//==============================================================
// 五盘阻尼器上下料主流程
//
// 一个bStart上升沿按Tray启动时冻结的物理层计划处理料盘，每盘4行×6列。
//
// 当前测试版本：
// 1. DamperX、DamperY在同一扫描周期启动；
// 2. 分别锁存X、Y完成信号，全部到位后继续；
// 3. 夹爪步骤直接通过；
// 4. 转台使用轴8在0°/180°之间绝对位置交替运动；
// 5. 夹紧轴使用位置模式模拟夹紧；
// 6. 调整过程由FB_TurntableProcess使用3秒TON模拟；
// 7. 换盘过程使用3秒TON模拟；
// 8. XY/Z/Rotation独立监督；统一Process Fault接入整机Stop链。
//==============================================================

FUNCTION_BLOCK FB_DamperProcess

VAR_INPUT
	
	bGripperActionDone  : BOOL; // 上一扫描至本扫描的动作FB结果
	bGripperActionError : BOOL;
    bGripperCloseTargetReachedWithoutGrip : BOOL;
    bGripperActionReady : BOOL; // Action Idle且Manager/Control均已释放
    // FALSE变为TRUE时启动完整五盘循环。
    bStart : BOOL;

    // 调试时产生上升沿，重新计算料位、备料位和缓冲位坐标。
    // 正常自动运行期间不要触发。
    bReinitializeCoordinates : BOOL;
	
	// 来自转台协调FB；由于MAIN先调用本FB，这里读取上一扫描周期状态。
    stTurntableStatus : ST_DamperTurntableStatus;
	// 当前料盘已经到达阻尼器取料位置。
	bTrayAtDamperPosition : BOOL;
	
	// 一次换盘已经完成，新料盘到达工作位置。
	// 保持到本FB撤销bTrayChangeRequest。
	bTrayChangeDone : BOOL;
	
	// 当前位于阻尼器工作位置的实际料盘层号。
	nTrayAtDamperLayer : INT;
    bCurrentTrayIsLastPlanned : BOOL; // Tray转接：当前工作位置料盘是固定计划最终盘
	// TRUE：立即中止本轮阻尼器自动流程。
	// 不清空料位、备料位、调整位和缓冲位物料状态。
	bAbort : BOOL;
    bReset : BOOL; // 复用整机故障复位
	// TRUE表示整机准备FB已经完成Z=110、XY=(1,1)、Rotation=0。
	bMachinePrepared : BOOL;
END_VAR

VAR_IN_OUT
    stAxisX : ST_AxisInterface; // DamperX：行方向
    stAxisY : ST_AxisInterface; // DamperY：列方向
    stAxisZ : ST_AxisInterface; // DamperZ：升降方向
	
	// 阻尼器夹爪旋转轴，对应统一轴数组第6轴。
    stAxisRotation : ST_AxisInterface;
END_VAR

VAR_OUTPUT
    bError : BOOL;
    uiErrorAxis : UINT;
    udiErrorCode : UDINT;
    bBusy : BOOL;
    bDone : BOOL;
    bCurrentTrayDone : BOOL;
    bTrayChangeRequest : BOOL;
    bInitialized : BOOL;
	
    //==========================================================
    // Damper三轴自动流程启动预定位完成
    //
    // TRUE表示：
    // 1. DamperZ已经位于110mm安全高度；
    // 2. DamperX/Y已经位于(1,1)料位上方；
    // 3. Tray机构可以开始取第一盘。
    //==========================================================
    bPrePositionDone : BOOL;

    // 最近一次螺钉角度视觉事务诊断。
    bVisionFault : BOOL;
    // 为兼容现有监控符号保留；本版本不再生成或使用Fallback结果。
    bVisionFallbackUsed : BOOL;
    eVisionError : E_VisionError := E_VisionError.None;

    // 发送给FB_TurntableProcess的保持型请求。
    stTurntableInput : ST_DamperTurntableInput;
    // 最近一次完成调整的料盘编号。
    nLastCompletedTray : INT;

    nCurrentTray   : INT;
    nCurrentRow    : INT;
    nCurrentColumn : DINT;

//==============================================================
// 上一件阻尼器的原始取料位置
//
// 用途：
// 1. 阻尼器取走后，原料位临时显示Adjusting；
// 2. 阻尼器放到其他实际位置后，将仍为Adjusting的原料位清空；
// 3. 如果原料位已经被其他合格品占用，则不能错误清空。
//==============================================================
	nPreviousSourceTray   : INT;
	nPreviousSourceRow    : INT;
	nPreviousSourceColumn : DINT;

    eCurrentStep : E_DamperProcessStep;
    eTakeStep    : E_DamperTakeStep;
    ePlaceStep   : E_DamperPlaceStep;

    // 当前工作位置料盘的数据。
    aSlots : A_DamperSlotGrid;

    // 转台两个位置及最终缓冲位的内容状态。
    eTransferPositionState   : E_DamperSlotState;
    eAdjustmentPositionState : E_DamperSlotState;
    eBufferPositionState     : E_DamperSlotState;

    // 公共工作位置，单位mm。
    fTrayPickZ     : LREAL;
    fTraySafeZ     : LREAL;
    fTransferX     : LREAL;
    fTransferY     : LREAL;
    fTransferPickZ : LREAL;
    fTransferSafeZ : LREAL;
    fBufferX       : LREAL;
    fBufferY       : LREAL;
    fBufferPickZ   : LREAL;
    fBufferSafeZ   : LREAL;
	
	bGripperActionExecute : BOOL; // 给COM3动作FB的保持型请求
	eGripperActionCommand : E_GripperCommand;
    bGripperAllowCloseTargetWithoutGrip : BOOL;
END_VAR

VAR
    trigStart : R_TRIG;
    fbXYMotionTimeout : TON;
    fbZMotionTimeout : TON;
    fbRotationMotionTimeout : TON;
    trigReinitializeCoordinates : R_TRIG;
	
    //==========================================================
    // 料盘坐标参数
    //==========================================================





    //==========================================================
    // Z轴参数
    //==========================================================

	//==========================================================
	// Z轴统一抬升绝对位置
	//
	// 所有XY运动前，以及取放料完成后，Z轴均抬升到110mm。
	// 该位置是实际测量确认的安全位置，不再进行高度计算。
	//==========================================================

	
	//==========================================================
	// 转台备料位实测绝对坐标，单位mm
	//==========================================================


	
	
	//==========================================================
	// 最终缓冲位1绝对坐标
	//
	// 当前为临时模拟值。
	// 实测完成后只修改以下三个参数。
	//==========================================================



	
    //==========================================================
    // 测试运动参数
    //==========================================================




    // 判断某根XY轴是否已经在目标位置。


		
    //==========================================================
    // 主流程内部变量
    //==========================================================
    bCoordinatesInitialized : BOOL;
    bPreviousPartAvailable  : BOOL;
    // 单槽位内部结果：只推进搜索，不代表实际取料成功。
    bTakeSkippedNoScrew : BOOL;
    bTakeSkippedEmptySlot : BOOL; // 物理空位已Open并回安全Z，独立于视觉Skip

    fCurrentSlotX : LREAL;
    fCurrentSlotY : LREAL;

    //==========================================================
    // XY并行运动内部状态
    //==========================================================
    bXYCommandIssued : BOOL;
    bXDoneLatched    : BOOL;
    bYDoneLatched    : BOOL;

    //==========================================================
    // Z轴运动内部状态
    //==========================================================
    bZCommandIssued : BOOL;
    bZDoneLatched   : BOOL;
	
	bWaitingTrayResult : BOOL;//等待料盘更换完成
    nTrayAwaitingResult : INT;//
    bStartPending : BOOL;//开始信号
	
	// 转台后的并行流程锁存。
	bPreviousPlaceDone       : BOOL;
	bExchangeCompleteLatched : BOOL;
	
	
	//==============================================================
	// 取料前相机检测位置参数
	//
	// 相机位于夹爪Y正方向90mm，因此相机对准阻尼器时：
	// 轴Y目标位置 = 阻尼器Y位置 - 90mm。
	//==============================================================


	
	// 当前检测高度与统一安全高度相同。

	
	
	//==============================================================
	// PLC相机检测模拟参数
	//==============================================================
	
	// 每个阻尼器到达相机位置后等待2秒。

	
	// 模拟相机返回机械零点坐标系下的绝对角度。

	
	
	//==============================================================
	// DamperRotation临时运动参数
	//
	// 单位应与DamperRotation NC轴缩放一致，当前按照“度”使用。
	//==============================================================



	
	// 修正角绝对值小于该值时，不发送旋转命令。

	
	//==============================================================
	// 二维码扫描绝对角度参数
	//
	// XY到达转台备料位后，DamperZ保持在110mm，
	// DamperRotation绝对运动到“相机角度+扫码偏移角”。
	// 当前使用旋转完成作为二维码扫描成功条件。
	//==============================================================
	//==============================================================
	// 相机检测与旋转运行变量
	//==============================================================
	
	// 螺钉角度业务视觉封装；内部拥有独立FB_VisionRequest实例。
	fbScrewAngleVision : FB_ScrewAngleVision;
	
	// 相机对准当前阻尼器时，DamperXY的目标位置。
	fCurrentVisionX : LREAL;
	fCurrentVisionY : LREAL;
	
	// 锁存原始检测角度、Python给出的机械修正量和本件实际机械基准角度。
	fDetectedAngleLatched   : LREAL;
	fCorrectionAngleLatched : LREAL;
	fRotationBaseAngle      : LREAL;
	fScanTargetAngle        : LREAL;
	bRotationCorrectionRequired : BOOL;
	
	// 防止每扫描周期重复发送DamperRotation绝对运动命令。
	bRotationCommandIssued : BOOL;
	
	//==============================================================
	// 取料后Z轴抬升与DamperRotation并行运动完成锁存
	//
	// 两根轴的完成信号可能出现在不同PLC扫描周期，
	// 因此必须分别锁存，不能直接将两个bDone进行AND判断。
	//==============================================================
	
	// 夹紧后：Z轴抬升与Rotation到相机角度的完成锁存。
	bCameraLiftZDoneLatched    : BOOL;
	bCameraRotationDoneLatched : BOOL;
	
	// 放料后：Z轴抬升、转台换位与Rotation回零的完成锁存。
	bResetLiftZDoneLatched     : BOOL;
	bResetTurntableDoneLatched : BOOL;
	bResetRotationDoneLatched  : BOOL;
END_VAR

//==============================================================
// 1. 更新输入上升沿
//==============================================================
trigStart(CLK := bStart);

trigReinitializeCoordinates(
    CLK := bReinitializeCoordinates
);

bGripperActionExecute := FALSE;
eGripperActionCommand := E_GripperCommand.None;
bGripperAllowCloseTargetWithoutGrip := FALSE;

// 机械流程只保持请求并消费统一结果；Simulation延时和ADS握手
// 均封装在FB_ScrewAngleVision中。
fbScrewAngleVision(
    bExecute := bBusy
                AND (eCurrentStep = E_DamperProcessStep.TakeCurrentDamper)
                AND (eTakeStep = E_DamperTakeStep.AcquireVisionResult),
    bCancel := bAbort OR bReset
);

//==============================================================
// 外部中止优先级最高
//==============================================================
IF bReset THEN
    bError := FALSE;
    uiErrorAxis := 0;
    udiErrorCode := TO_UDINT(E_DamperErrorCode.None);
    bVisionFault := FALSE;
    eVisionError := E_VisionError.None;
END_IF;

IF bAbort OR bReset THEN
    M_AbortProcess(
        ioAxisX := stAxisX,
        ioAxisY := stAxisY,
        ioAxisZ := stAxisZ,
        ioAxisRotation := stAxisRotation
    );

    RETURN;
END_IF;


IF trigStart.Q AND NOT bError THEN
    // 锁存一次完整五盘流程启动请求。
    bStartPending := TRUE;

    // 新一轮流程必须重新执行Damper三轴预定位。
    // 防止上一轮残留的TRUE让Tray机构提前启动。
    bPrePositionDone := FALSE;
END_IF;


	// 当前测试阶段让转台协调FB一直保持使能，先完成0°和松开位置初始化。
	// 实机后可改为系统自动模式许可。
	stTurntableInput.bEnable := bStart
								OR bStartPending
								OR bBusy;
	stTurntableInput.bAdjustmentAccepted := FALSE;
	stTurntableInput.bAdjustmentDone := FALSE;
	// 最终质量只由FB_AdjustmentProcess经协调器写入，Damper不再提供固定合格值。
	stTurntableInput.bAdjustmentQualified := FALSE;
	stTurntableInput.bTransferCaptureOK := TRUE;
	stTurntableInput.bAdjustmentCaptureOK := TRUE;
	stTurntableInput.bReset := FALSE;
//==============================================================
// 2. 首次调用或调试命令触发时初始化坐标
//
// 重新初始化坐标不会修改生产状态。
//==============================================================
IF
    (NOT bCoordinatesInitialized)
    OR
    (
        trigReinitializeCoordinates.Q
        AND NOT bBusy
    )
THEN
    M_InitializeDamperCoordinates();
    bCoordinatesInitialized := TRUE;
END_IF;


//==============================================================
// 3. 模拟换盘定时器
//
// 只有进入WaitTrayChange时定时器才开始计时。
// 离开该步骤后自动复位。
//==============================================================

//==============================================================
// 4. 清除单周期输出
//==============================================================
bCurrentTrayDone := FALSE;

// 第24件可能在更换料盘、甚至下一盘第1件取料期间完成调整，
// 所以该检测必须独立于主CASE每周期执行。
IF
    bWaitingTrayResult
    AND
    (
        (
            eAdjustmentPositionState
            = E_DamperSlotState.Qualified
        )
        OR
        (
            eAdjustmentPositionState
            = E_DamperSlotState.Unqualified
        )
    )
THEN
    bCurrentTrayDone := TRUE;
    nLastCompletedTray := nTrayAwaitingResult;
    bWaitingTrayResult := FALSE;
END_IF;

//==============================================================
// 5. 自动运行期间清除上一周期运动命令
//
// 各运动辅助Method会在需要时重新生成
// 一个PLC周期的bMoveAbs命令脉冲。
//==============================================================
IF bBusy THEN
    stAxisX.AutoCmd.bMoveAbs := FALSE;
    stAxisY.AutoCmd.bMoveAbs := FALSE;
    stAxisZ.AutoCmd.bMoveAbs := FALSE;

    // DamperRotation只使用绝对位置运动。
    stAxisRotation.AutoCmd.bMoveAbs := FALSE;
END_IF;

//==============================================================
// 6. 换盘请求
//
// 进入WaitTrayChange后保持TRUE，离开后恢复FALSE。
//==============================================================
bTrayChangeRequest :=
    eCurrentStep
    = E_DamperProcessStep.WaitTrayChange;

//==============================================================
// 7. 五盘阻尼器上下料主流程
//==============================================================
CASE eCurrentStep OF

    //==========================================================
	// 空闲：等待自动启动上升沿
	//==========================================================
	E_DamperProcessStep.Idle:
		bBusy := FALSE;
		bDone := FALSE;
		bTrayChangeRequest := FALSE;
		bPrePositionDone := FALSE;
	
		bPreviousPlaceDone := FALSE;
		bExchangeCompleteLatched := FALSE;
	
		stTurntableInput.bExchangeRequest := FALSE;
		stTurntableInput.bNoMorePartsToLoad := FALSE;
		stTurntableInput.bFinalUnloadDone := FALSE;
	
		bWaitingTrayResult := FALSE;
		nTrayAwaitingResult := 0;
	
		nLastCompletedTray := 0;
		nCurrentTray := 0;
		nCurrentRow := 0;
		nCurrentColumn := 0;
	
		bPreviousPartAvailable := FALSE;
		bTakeSkippedNoScrew := FALSE;
		bTakeSkippedEmptySlot := FALSE;
	
		// 清除上一件阻尼器来源位置。
		nPreviousSourceTray := 0;
		nPreviousSourceRow := 0;
		nPreviousSourceColumn := 0;
	
		// 新一轮流程开始时，转台两个位置和缓冲位均按空处理。
		eTransferPositionState :=
			E_DamperSlotState.Empty;
	
		eAdjustmentPositionState :=
			E_DamperSlotState.Empty;
	
		eBufferPositionState :=
			E_DamperSlotState.Empty;
	
		eTakeStep := E_DamperTakeStep.Idle;
		ePlaceStep := E_DamperPlaceStep.Idle;
	
		//======================================================
		// 先启动Damper三轴预定位。
		//
		// 此处不再等待第一盘到位，也不等待转台初始化完成。
		// Damper预定位与转台初始化可以同时执行。
		//======================================================
		IF
			bStartPending
			AND bCoordinatesInitialized
	
			// 三根轴必须可以接受绝对位置运动命令。
			AND stAxisX.State.bReady
			AND stAxisY.State.bReady
			AND stAxisZ.State.bReady
			AND stAxisRotation.State.bReady
		THEN
			bStartPending := FALSE;
	
			// 清除运动Method内部的命令和完成锁存。
			M_ResetMotionHelpers(
				ioAxisX := stAxisX,
				ioAxisY := stAxisY,
				ioAxisZ := stAxisZ,
				ioAxisRotation := stAxisRotation
			);	
			// 第一盘进入工作位置后，默认24个位置都有未调整阻尼器。
			M_ResetDamperSlotStates();
	
			nCurrentTray := 0; // 第一盘到位时再锁存真实物理层号
			nCurrentRow := 1;
			nCurrentColumn := 1;
	
			bBusy := TRUE;
	
			// 第一步必须先让DamperZ运动到110mm安全高度。
			IF bMachinePrepared THEN
				// 整机准备FB已经完成预定位，直接等待第一盘。
				bPrePositionDone := TRUE;
				eCurrentStep := E_DamperProcessStep.WaitFirstTray;
			ELSE
				// 保留独立调试时的兼容入口。
				eCurrentStep := E_DamperProcessStep.InitializeSafeZ;
			END_IF;
		END_IF;

	//==========================================================
	// 自动启动预定位第1步：DamperZ先到110mm安全位置
	//==========================================================
	E_DamperProcessStep.InitializeSafeZ:
		bBusy := TRUE;
		bPrePositionDone := FALSE;
	
		IF M_MoveZAbsolute(
			fTargetZ := fTraySafeZ,
			ioAxisZ := stAxisZ
		) THEN
			// Z轴确认到达110mm后，才允许X/Y移动。
			eCurrentStep :=
				E_DamperProcessStep.InitializeXYFirstSlot;
		END_IF;
	
	
	//==========================================================
	// 自动启动预定位第2步：DamperX/Y到(1,1)上方
	//==========================================================
	E_DamperProcessStep.InitializeXYFirstSlot:
		bBusy := TRUE;
		bPrePositionDone := FALSE;
	
		// 直接读取初始化后的(1,1)实际坐标，
		// 后续修改料位基准坐标时不需要修改本流程。
		fCurrentSlotX :=
			aSlots[1, 1].fXPosition;
	
		fCurrentSlotY :=
			aSlots[1, 1].fYPosition;
	
		// 两根独立轴在同一扫描周期发送绝对运动命令，
		// 分别确认到位后才继续。
		IF M_MoveXYParallel(
			fTargetX := fCurrentSlotX,
			fTargetY := fCurrentSlotY,
			ioAxisX := stAxisX,
			ioAxisY := stAxisY
		) THEN
			// 三轴预定位完成，允许Tray机构开始运动。
			bPrePositionDone := TRUE;
	
			eCurrentStep :=
				E_DamperProcessStep.WaitFirstTray;
		END_IF;
	
	
	//==========================================================
	// 自动启动预定位第3步：等待第一盘和转台准备完成
	//==========================================================
	E_DamperProcessStep.WaitFirstTray:
		bBusy := TRUE;
	
		// 保持TRUE，让Tray流程能够可靠收到允许启动信号。
		bPrePositionDone := TRUE;
	
		IF
			// 第一盘已经由Tray机构送到阻尼器取料位置。
			bTrayAtDamperPosition
            AND (nTrayAtDamperLayer >= LOWER_BOUND(GVL_PositionConfig.stTray.aLayer, 1))
            AND (nTrayAtDamperLayer <= UPPER_BOUND(GVL_PositionConfig.stTray.aLayer, 1))
	
			// 转台初始化已经完成：
			// 夹紧轴处于松开位置，转台位于初始位置。
			AND stTurntableStatus.bReady
	
			// 三根Damper轴当前仍然可以继续执行运动。
			AND stAxisX.State.bReady
			AND stAxisY.State.bReady
			AND stAxisZ.State.bReady
			AND stAxisRotation.State.bReady
		THEN
			nCurrentTray := nTrayAtDamperLayer;
			// 第一盘到位后进入原有第一件取料流程。
			// M_TakeDamper中的安全Z和XY检查会因为已经到位而直接通过，
			// 随后DamperZ下降到第一料位取料高度。
			eCurrentStep :=
				E_DamperProcessStep.TakeCurrentDamper;
		END_IF;

    //==========================================================
    // 从当前料盘料位取出未调整阻尼器并放到转台备料位
    //==========================================================
    E_DamperProcessStep.TakeCurrentDamper:
        fCurrentSlotX :=
            aSlots[nCurrentRow, nCurrentColumn].fXPosition;

        fCurrentSlotY :=
            aSlots[nCurrentRow, nCurrentColumn].fYPosition;
		// 尚未开始取料时，必须确认转台备料位允许放入。
		// 一旦M_TakeDamper内部流程已经启动，则继续执行，不能中途暂停。
		IF
			(eTakeStep <> E_DamperTakeStep.Idle)
			OR stTurntableStatus.bReadyForTransferLoad
		THEN
			IF M_TakeDamper(
				fSourceX := fCurrentSlotX,
				fSourceY := fCurrentSlotY,
			
				ioAxisX := stAxisX,
				ioAxisY := stAxisY,
				ioAxisZ := stAxisZ,
			
				// 新增DamperRotation轴。
				ioAxisRotation := stAxisRotation
			) THEN				
				// 当前Method返回时：
				// 1. 阻尼器已经放入转台备料位；
				// 2. Z轴已经回到安全高度；
				// 3. 转台已经完成下一工位旋转；
				// 4. DamperRotation已经绝对回到机械零点。
				aSlots[nCurrentRow, nCurrentColumn].eState :=
					E_DamperSlotState.Empty;
			
				eCurrentStep := E_DamperProcessStep.RotateTurntable;
			ELSIF bTakeSkippedNoScrew THEN
				// M_TakeDamper仍返回FALSE：Skip没有任何真实取料副作用。
				// eTakeStep已退出AcquireVisionResult；下一扫描bExecute=FALSE
				// 复位本笔视觉事务，下一槽位重新到相机位后才发起新请求。
				bTakeSkippedNoScrew := FALSE;
				bTakeSkippedEmptySlot := FALSE;

				IF nCurrentColumn < UPPER_BOUND(aSlots, 2) THEN
					nCurrentColumn := nCurrentColumn + 1;
				ELSIF nCurrentRow < UPPER_BOUND(aSlots, 1) THEN
					nCurrentColumn := LOWER_BOUND(aSlots, 2);
					nCurrentRow := nCurrentRow + 1;
				ELSE
					// 盘尾Skip只结束搜索；保留最后一次真实取料的来源与在途状态。
					// 仅本盘真实尾件需要登记调整结果；全盘Skip不创建等待工件。
					IF bPreviousPartAvailable AND (nPreviousSourceTray = nCurrentTray) THEN
						bWaitingTrayResult := TRUE;
						nTrayAwaitingResult := nCurrentTray;
					END_IF;

					IF NOT bCurrentTrayIsLastPlanned THEN
						eCurrentStep := E_DamperProcessStep.WaitTrayChange;
					ELSIF bPreviousPartAvailable THEN
						// 最终计划盘仍有真实尾件：使用原最终收尾路径。
						eCurrentStep := E_DamperProcessStep.FinalWaitAdjustment;
					ELSE
						// 无真实在途件：不等待不存在的调整结果、不请求空转。
						eCurrentStep := E_DamperProcessStep.Completed;
					END_IF;
				END_IF;
            ELSIF bTakeSkippedEmptySlot THEN
                // 仅Open Done且安全Z真正到位后产生；物料Empty已由取料层确认。
                // 不返回真实取料成功，不改最后真实工件的来源或在途状态。
                bTakeSkippedEmptySlot := FALSE;
				IF nCurrentColumn < UPPER_BOUND(aSlots, 2) THEN
					nCurrentColumn := nCurrentColumn + 1;
				ELSIF nCurrentRow < UPPER_BOUND(aSlots, 1) THEN
					nCurrentColumn := LOWER_BOUND(aSlots, 2);
					nCurrentRow := nCurrentRow + 1;
				ELSE
					// 盘尾Skip只结束搜索；保留最后一次真实取料的来源与在途状态。
					// 仅本盘真实尾件需要登记调整结果；全盘Skip不创建等待工件。
					IF bPreviousPartAvailable AND (nPreviousSourceTray = nCurrentTray) THEN
						bWaitingTrayResult := TRUE;
						nTrayAwaitingResult := nCurrentTray;
					END_IF;

					IF NOT bCurrentTrayIsLastPlanned THEN
						eCurrentStep := E_DamperProcessStep.WaitTrayChange;
					ELSIF bPreviousPartAvailable THEN
						// 最终计划盘仍有真实尾件：使用原最终收尾路径。
						eCurrentStep := E_DamperProcessStep.FinalWaitAdjustment;
					ELSE
						// 无真实在途件：不等待不存在的调整结果、不请求空转。
						eCurrentStep := E_DamperProcessStep.Completed;
					END_IF;
				END_IF;
			END_IF;
		END_IF;


	//==========================================================
	// 兼容保留步骤
	//
	// 调整结果现在完全由FB_TurntableProcess管理，
	// 本步骤不得再直接修改eAdjustmentPositionState。
	//==========================================================
	E_DamperProcessStep.WaitPreviousAdjustment:
		stTurntableInput.bExchangeRequest := TRUE;
	
		eCurrentStep :=
			E_DamperProcessStep.RotateTurntable;


	//==========================================================
	// 模拟转台旋转180°
	//
	// 进入该步骤后等待3秒。
	// 定时完成才认为转台到位，然后交换两个物理位置状态。
	//==========================================================
	E_DamperProcessStep.RotateTurntable:
		// bExchangeDone可能在机械手放料完成之前出现，因此需要锁存。
		IF stTurntableStatus.bExchangeDone THEN
			bExchangeCompleteLatched := TRUE;
		END_IF;
	
		IF bPreviousPartAvailable THEN
			// 转台物理到位后立即开始取回上一件。
			// 此时FB_TurntableProcess会同时启动夹紧轴。
			IF stTurntableStatus.bRotationDone THEN
				eCurrentStep :=
					E_DamperProcessStep.PlacePreviousDamper;
			END_IF;
	
		ELSE
			// 第一盘第一件旋转后，取回位置为空。
			// 不需要DamperZ取料，只等待夹紧完成。
			IF bExchangeCompleteLatched THEN
				stTurntableInput.bExchangeRequest := FALSE;
				bExchangeCompleteLatched := FALSE;
	
				eCurrentStep :=
					E_DamperProcessStep.FinishCurrentSlot;
			END_IF;
		END_IF;

    //==========================================================
    // 将上一件已调整阻尼器放入当前刚取空的料位
    //
    // X、Y作为Method输入参数。
    // 如果将来需要放回上一件原始位置，只需在此处改为
    // 上一件原始料位的X、Y，不需要修改Method内部代码。
    //==========================================================
    E_DamperProcessStep.PlacePreviousDamper:
		// 夹紧轴可能先完成，因此持续锁存转台完整交换完成状态。
		IF stTurntableStatus.bExchangeDone THEN
			bExchangeCompleteLatched := TRUE;
		END_IF;
	
		// Damper机械手支路尚未完成时，持续执行取回和放料Method。
		IF NOT bPreviousPlaceDone THEN
			IF M_PlaceDamper(
				fTargetX := fCurrentSlotX,
				fTargetY := fCurrentSlotY,
				fTargetZ := fTrayPickZ,
				fTargetSafeZ := fTraySafeZ,
				ioAxisX := stAxisX,
				ioAxisY := stAxisY,
				ioAxisZ := stAxisZ
			) THEN
				// 如果上一件的原始位置仍为Adjusting，则清空。
				IF
					(nPreviousSourceTray = nCurrentTray)
					AND
					(
						(nPreviousSourceRow <> nCurrentRow)
						OR
						(nPreviousSourceColumn <> nCurrentColumn)
					)
					AND
					(
						aSlots[
							nPreviousSourceRow,
							nPreviousSourceColumn
						].eState
						= E_DamperSlotState.Adjusting
					)
				THEN
					aSlots[
						nPreviousSourceRow,
						nPreviousSourceColumn
					].eState :=
						E_DamperSlotState.Empty;
				END_IF;
	
				// 实际放入位置显示调整结果。
				aSlots[nCurrentRow, nCurrentColumn].eState :=
					eTransferPositionState;
	
				// 取回位已经被机械手取空。
				eTransferPositionState :=
					E_DamperSlotState.Empty;
	
				bPreviousPlaceDone := TRUE;
			END_IF;
		END_IF;
	
		//==========================================================
		// 两个并行支路都完成后，本轮交换才结束：
		//
		// 1. Damper机械手已经把上一件放入实际料位；
		// 2. 夹紧轴已经完成夹紧，转台FB发出bExchangeDone。
		//==========================================================
		IF
			bPreviousPlaceDone
			AND bExchangeCompleteLatched
		THEN
			stTurntableInput.bExchangeRequest := FALSE;
	
			bPreviousPlaceDone := FALSE;
			bExchangeCompleteLatched := FALSE;
	
			eCurrentStep :=
				E_DamperProcessStep.FinishCurrentSlot;
		END_IF;


    //==========================================================
    // 当前料位处理完成，计算下一个料位
    //==========================================================
    E_DamperProcessStep.FinishCurrentSlot:
		// 当前送入调整位的阻尼器，将在下一次转台旋转后被取回。
		bPreviousPartAvailable := TRUE;
		
		// 保存当前阻尼器的原始取料位置。
		// 下一次执行PlacePreviousDamper时，这些变量代表被放回阻尼器的来源。
		nPreviousSourceTray := nCurrentTray;
		nPreviousSourceRow := nCurrentRow;
		nPreviousSourceColumn := nCurrentColumn;
		
        IF nCurrentColumn < UPPER_BOUND(aSlots, 2) THEN
            // 同一行内，列号增加。
            // 下一次取料时DamperX目标不变，只有DamperY需要运动。
            nCurrentColumn := nCurrentColumn + 1;

            eCurrentStep :=
                E_DamperProcessStep.TakeCurrentDamper;

        ELSIF nCurrentRow < UPPER_BOUND(aSlots, 1) THEN
            // 当前行结束：
            // DamperY回第1列，DamperX进入下一行。
            //
            // 两轴会在同一个扫描周期启动，
            // 不进行直线插补。
            nCurrentColumn := 1;
            nCurrentRow := nCurrentRow + 1;

            eCurrentStep :=
                E_DamperProcessStep.TakeCurrentDamper;

        ELSE
            // 当前盘第24件已经进入调整位，
			IF (nCurrentRow = UPPER_BOUND(aSlots, 1)) AND (nCurrentColumn = UPPER_BOUND(aSlots, 2)) THEN
				// 记录是哪一盘的第24件正在等待调整结果。
				bWaitingTrayResult := TRUE;
				nTrayAwaitingResult := nCurrentTray;
			END_IF;
            // 第23件已经放入当前盘第24个空料位。
            IF NOT bCurrentTrayIsLastPlanned THEN
                // 方案B：
                // 第24件处于调整位期间，开始模拟更换料盘。
                eCurrentStep :=
                    E_DamperProcessStep.WaitTrayChange;
            ELSE
                // 最终计划盘不再更换新料盘。
                eCurrentStep :=
                    E_DamperProcessStep.FinalWaitAdjustment;
            END_IF;
        END_IF;


    //==========================================================
    // 模拟更换料盘
    //
    // 方案B：
    // 第24件在调整位调整的同时，料盘进行更换。
    //
    // 当前版本：
    // 1. 调整直接判定合格；
    // 2. 换盘使用3秒定时器；
    // 3. 定时完成后初始化下一盘24个料位。
    //
    // 后续联动FB_TrayProcess时：
    // 1. 保留bTrayChangeRequest；
    // 2. 删除或旁路fbSimulatedTrayChange.Q；
    // 3. 改为等待实际bTrayChangeDone信号。
    //==========================================================
	//==========================================================
	// 模拟换盘
	//
	// 只等待料盘更换完成，不再等待上一盘第24件调整完成。
	// 允许新盘第1件先进入空的备料位。
	//==========================================================
	E_DamperProcessStep.WaitTrayChange:
		//==========================================================
		// 等待下一盘真正到达阻尼器取料位置
		//
		// 同时判断层号，防止旧料盘尚未离开时
		// bTrayAtDamperPosition仍为TRUE而造成误判。
		//==========================================================
		IF
			bTrayChangeDone
			AND bTrayAtDamperPosition
            AND (nTrayAtDamperLayer > nCurrentTray)
            AND (nTrayAtDamperLayer <= UPPER_BOUND(GVL_PositionConfig.stTray.aLayer, 1))
		THEN
			nCurrentTray := nTrayAtDamperLayer;
			nCurrentRow := 1;
			nCurrentColumn := 1;
	
			// 从现在开始，aSlots表示新到达的料盘。
			M_ResetDamperSlotStates();
	
			// 保留此前真实取料建立的在途状态；全盘Skip不能凭换盘创建工件。
			bTakeSkippedNoScrew := FALSE;
			bTakeSkippedEmptySlot := FALSE;
	
			eCurrentStep :=
				E_DamperProcessStep.TakeCurrentDamper;
		END_IF;


	//==========================================================
	// 等待最终计划盘第24件调整完成
	//==========================================================
	E_DamperProcessStep.FinalWaitAdjustment:
		IF
			(
				eAdjustmentPositionState
				= E_DamperSlotState.Qualified
			)
			OR
			(
				eAdjustmentPositionState
				= E_DamperSlotState.Unqualified
			)
		THEN
			// 最终计划盘第24件之后不再有下一件。
			stTurntableInput.bNoMorePartsToLoad := TRUE;
			stTurntableInput.bExchangeRequest := TRUE;
			eCurrentStep := E_DamperProcessStep.FinalRotateTurntable;
		END_IF;


 	//==========================================================
	// 最终计划盘第24件调整完成后，模拟转台旋转180°
	//==========================================================
	E_DamperProcessStep.FinalRotateTurntable:
		IF
			stTurntableStatus.bExchangeDone
			AND stTurntableStatus.bFinalUnloadRequest
		THEN
			stTurntableInput.bExchangeRequest := FALSE;
			eCurrentStep :=
				E_DamperProcessStep.PlaceFinalDamperToBuffer;
		END_IF;


    //==========================================================
	// 将最终计划盘第24件从转台取回位搬到缓冲位1
	//==========================================================
	E_DamperProcessStep.PlaceFinalDamperToBuffer:
		IF M_PlaceDamper(
			fTargetX := fBufferX,
			fTargetY := fBufferY,
			fTargetZ := fBufferPickZ,
			fTargetSafeZ := fBufferSafeZ,
			ioAxisX := stAxisX,
			ioAxisY := stAxisY,
			ioAxisZ := stAxisZ
		) THEN
			// M_PlaceDamper返回TRUE时，阻尼器已经实际放到缓冲位，
			// 并且Z轴已经回到缓冲位安全高度。
	
			// 缓冲位记录实际放入物料的检测结果。
			eBufferPositionState :=
				eTransferPositionState;
	
			// 阻尼器已经离开转台取回位。
			eTransferPositionState :=
				E_DamperSlotState.Empty;
	
			// 最终搬运完成保持型应答。
			stTurntableInput.bFinalUnloadDone := TRUE;
	
			bPreviousPartAvailable := FALSE;
	
			eCurrentStep :=
				E_DamperProcessStep.Completed;
		END_IF;
		//==========================================================
		// 五盘流程完成
		//
		// bDone采用锁存方式保持，直到产生下一次启动上升沿。
		// 因此bStart可以是短脉冲，不需要一直保持TRUE。
		//==========================================================
		E_DamperProcessStep.Completed:
			// 等转台撤销最终取回请求后，完整流程才算结束。
			IF NOT stTurntableStatus.bFinalUnloadRequest THEN
				// 四相握手最后一步：
				// 请求方确认对方已撤销Request后，再撤销Done。
				stTurntableInput.bFinalUnloadDone := FALSE;
				stTurntableInput.bNoMorePartsToLoad := FALSE;
		
				bBusy := FALSE;
				bDone := TRUE;
				bTrayChangeRequest := FALSE;
			END_IF;
		
			// 下一次bStart上升沿已经在程序顶部锁存为bStartPending。
			// 清除上一次完成状态并回到Idle，下一扫描周期重新启动。
			IF bDone AND bStartPending THEN
				bDone := FALSE;
		
				eCurrentStep :=
					E_DamperProcessStep.Idle;
			END_IF;


	//==========================================================
	// 螺钉视觉/运动失败锁存终态
	//
	// 不自动重试、不跳件、不回安全位；仅撤销自动命令和流程请求，
	// 保留bVisionFault/eVisionError，等待现有bAbort或系统复位处理。
	//==========================================================
	E_DamperProcessStep.Error:
        bTakeSkippedEmptySlot := FALSE;
		bBusy := FALSE;
		bDone := FALSE;
		bTrayChangeRequest := FALSE;
		bPrePositionDone := FALSE;

		eTakeStep := E_DamperTakeStep.Idle;
		ePlaceStep := E_DamperPlaceStep.Idle;

		bGripperActionExecute := FALSE;
		eGripperActionCommand := E_GripperCommand.None;
		bGripperAllowCloseTargetWithoutGrip := FALSE;

		stAxisX.AutoCmd.bMoveAbs := FALSE;
		stAxisY.AutoCmd.bMoveAbs := FALSE;
		stAxisZ.AutoCmd.bMoveAbs := FALSE;
		stAxisRotation.AutoCmd.bMoveAbs := FALSE;
		stAxisRotation.AutoCmd.bMoveRel := FALSE;

		stTurntableInput.bEnable := FALSE;
		stTurntableInput.bExchangeRequest := FALSE;
		stTurntableInput.bNoMorePartsToLoad := FALSE;
		stTurntableInput.bFinalUnloadDone := FALSE;


ELSE
    // 非法步骤直接回到Idle。
    // 当前版本不实现异常恢复。
    bBusy := FALSE;
    bDone := FALSE;
    bTrayChangeRequest := FALSE;

    eCurrentStep :=
        E_DamperProcessStep.Idle;

END_CASE;

// 子流程本扫描首次报错时，立即撤销全部请求；不改变物料状态。
IF bError THEN
    M_AbortProcess(
        ioAxisX := stAxisX,
        ioAxisY := stAxisY,
        ioAxisZ := stAxisZ,
        ioAxisRotation := stAxisRotation
    );
END_IF;

METHOD PRIVATE M_AbortProcess

VAR_IN_OUT
    ioAxisX        : ST_AxisInterface;
    ioAxisY        : ST_AxisInterface;
    ioAxisZ        : ST_AxisInterface;
    ioAxisRotation : ST_AxisInterface;
END_VAR
//==============================================================
// 1. 清除本流程产生的运动命令
//==============================================================
ioAxisX.AutoCmd.bMoveAbs := FALSE;
ioAxisX.AutoCmd.bMoveRel := FALSE;
ioAxisX.AutoCmd.bJogPos := FALSE;
ioAxisX.AutoCmd.bJogNeg := FALSE;

ioAxisY.AutoCmd.bMoveAbs := FALSE;
ioAxisY.AutoCmd.bMoveRel := FALSE;
ioAxisY.AutoCmd.bJogPos := FALSE;
ioAxisY.AutoCmd.bJogNeg := FALSE;

ioAxisZ.AutoCmd.bMoveAbs := FALSE;
ioAxisZ.AutoCmd.bMoveRel := FALSE;
ioAxisZ.AutoCmd.bJogPos := FALSE;
ioAxisZ.AutoCmd.bJogNeg := FALSE;

ioAxisRotation.AutoCmd.bMoveAbs := FALSE;
ioAxisRotation.AutoCmd.bMoveRel := FALSE;
ioAxisRotation.AutoCmd.bJogPos := FALSE;
ioAxisRotation.AutoCmd.bJogNeg := FALSE;

ioAxisX.AutoCmd.bTorqueControl := FALSE;
ioAxisY.AutoCmd.bTorqueControl := FALSE;
ioAxisZ.AutoCmd.bTorqueControl := FALSE;
ioAxisRotation.AutoCmd.bTorqueControl := FALSE;
//==============================================================
// 2. 复位运动辅助锁存
//==============================================================
M_ResetMotionHelpers(
    ioAxisX := ioAxisX,
    ioAxisY := ioAxisY,
    ioAxisZ := ioAxisZ,
    ioAxisRotation := ioAxisRotation
);

bWaitingTrayResult := FALSE;
bPreviousPlaceDone := FALSE;
bExchangeCompleteLatched := FALSE;
bStartPending := FALSE;

bRotationCommandIssued := FALSE;
bCameraLiftZDoneLatched := FALSE;
bCameraRotationDoneLatched := FALSE;
bResetLiftZDoneLatched := FALSE;
bResetTurntableDoneLatched := FALSE;
bResetRotationDoneLatched := FALSE;


//==============================================================
// 4. 撤销发往转台的全部请求
//
// stTurntableInput.bEnable=FALSE后，
// FB_TurntableProcess会进入现有的禁用复位分支。
//==============================================================
stTurntableInput.bEnable := FALSE;
stTurntableInput.bExchangeRequest := FALSE;
stTurntableInput.bNoMorePartsToLoad := FALSE;
stTurntableInput.bAdjustmentAccepted := FALSE;
stTurntableInput.bAdjustmentDone := FALSE;
stTurntableInput.bAdjustmentQualified := FALSE;
stTurntableInput.bFinalUnloadDone := FALSE;
stTurntableInput.bTransferCaptureOK := FALSE;
stTurntableInput.bAdjustmentCaptureOK := FALSE;
stTurntableInput.bReset := FALSE;


//==============================================================
// 5. 清除流程输出和握手
//==============================================================
bGripperActionExecute := FALSE;
eGripperActionCommand := E_GripperCommand.None;
bGripperAllowCloseTargetWithoutGrip := FALSE;
bTakeSkippedEmptySlot := FALSE;
bBusy := FALSE;
bDone := FALSE;
bCurrentTrayDone := FALSE;
bTrayChangeRequest := FALSE;
bPrePositionDone := FALSE;


//==============================================================
// 6. 状态机返回空闲
//==============================================================
IF bError THEN
    eCurrentStep := E_DamperProcessStep.Error;
ELSE
    eCurrentStep := E_DamperProcessStep.Idle;
END_IF;
eTakeStep := E_DamperTakeStep.Idle;
ePlaceStep := E_DamperPlaceStep.Idle;


//==============================================================
// 7. 有意保留的物料数据
//
// 不修改：
// aSlots
// eTransferPositionState
// eAdjustmentPositionState
// eBufferPositionState
// bPreviousPartAvailable及原料位索引
//
// 停止时物料可能正在夹爪或转台中，
// 当前版本由操作员确认并手动恢复现场。
//==============================================================
END_METHOD

//==============================================================
// 初始化24个料位坐标以及公共工作位置
//
// 本Method只修改坐标，不修改任何料位内容状态。
//==============================================================
METHOD PRIVATE M_InitializeDamperCoordinates

VAR
    nRow : DINT;
    nColumn : DINT;
END_VAR
//==============================================================
// 1. 初始化24个料位XY坐标
//==============================================================
FOR nRow := 1 TO UPPER_BOUND(aSlots, 1) DO
    FOR nColumn := 1 TO UPPER_BOUND(aSlots, 2) DO
        aSlots[nRow, nColumn].fXPosition :=
            GVL_PositionConfig.stDamper.stGrid.stOrigin.X
            + DINT_TO_LREAL(nRow - 1) * GVL_PositionConfig.stDamper.stGrid.fRowPitchX
            + GVL_PositionConfig.stDamper.stGrid.aSlotOffset[nRow, nColumn].X;

        aSlots[nRow, nColumn].fYPosition :=
            GVL_PositionConfig.stDamper.stGrid.stOrigin.Y
            + DINT_TO_LREAL(nColumn - 1) * GVL_PositionConfig.stDamper.stGrid.fColumnPitchY
            + GVL_PositionConfig.stDamper.stGrid.aSlotOffset[nRow, nColumn].Y;
    END_FOR
END_FOR;


	//==============================================================
	// 2. 料盘Z轴位置
	//==============================================================
	// 料盘取放绝对高度。
	fTrayPickZ := GVL_PositionConfig.stDamper.stGrid.fPickZ;
	
	// 料盘区域XY移动前统一抬升到110mm。
	fTraySafeZ := GVL_PositionConfig.stDamper.fSafeZ;

	//==============================================================
	// 3. 备料/取回位
	//==============================================================
	//==============================================================
	// 备料位使用实测绝对坐标
	//==============================================================
	fTransferX := GVL_PositionConfig.stDamper.stTransfer.X;
	fTransferY := GVL_PositionConfig.stDamper.stTransfer.Y;
	fTransferPickZ := GVL_PositionConfig.stDamper.stTransfer.Z;
	
	// 备料位取放完成后，同样抬升到固定110mm。
	fTransferSafeZ := GVL_PositionConfig.stDamper.fSafeZ;



	//==============================================================
	// 4. 最终缓冲位
	//
	// 当前临时坐标：
	// 缓冲位实测目标从GVL_PositionConfig.stDamper读取。
	//==============================================================
	// 最终缓冲位1直接使用绝对坐标。
	fBufferX := GVL_PositionConfig.stDamper.stBuffer.X;
	fBufferY := GVL_PositionConfig.stDamper.stBuffer.Y;
	fBufferPickZ := GVL_PositionConfig.stDamper.stBuffer.Z;
	
	// 所有取放完成后统一抬升到110mm。
	fBufferSafeZ := GVL_PositionConfig.stDamper.fSafeZ;
END_METHOD

//==============================================================
// DamperRotation统一绝对角度运动。
//
// 调用方只传入参数层提供或计算出的绝对目标角度，
// 本Method不读取当前角度进行目标累加。
//==============================================================
METHOD PRIVATE M_MoveRotationAbsolute : BOOL

VAR_INPUT
    fTargetAngle : LREAL;
    fVelocity : LREAL;
    fAcceleration : LREAL;
    fDeceleration : LREAL;
END_VAR

VAR_IN_OUT
    ioAxisRotation : ST_AxisInterface;
END_VAR
M_MoveRotationAbsolute := FALSE;
IF bError OR bAbort OR bReset THEN
    RETURN;
END_IF;
// 首次等待Ready也纳入本次运动计时；跨取料子步骤继续原Timer。
fbRotationMotionTimeout(IN := TRUE, PT := GVL_MotionConfig.stDamper.tMoveTimeout);

// 已在目标角度公差内时无需发令。
IF NOT bRotationCommandIssued THEN
    IF
        ABS(ioAxisRotation.Data.fActPosition - fTargetAngle)
        <= GVL_MotionConfig.stDamper.stRotation.fPositionTolerance
    THEN
        fbRotationMotionTimeout(IN := FALSE, PT := GVL_MotionConfig.stDamper.tMoveTimeout);
        M_MoveRotationAbsolute := TRUE;

    ELSIF ioAxisRotation.State.bReady THEN
        ioAxisRotation.AutoSet.Position.fAbsolutePosition := fTargetAngle;
        ioAxisRotation.AutoSet.Position.fVelocity := fVelocity;
        ioAxisRotation.AutoSet.Position.fAcceleration := fAcceleration;
        ioAxisRotation.AutoSet.Position.fDeceleration := fDeceleration;

        // 只产生一个PLC扫描周期的绝对运动命令脉冲。
        ioAxisRotation.AutoCmd.bMoveAbs := TRUE;
        bRotationCommandIssued := TRUE;
    ELSIF fbRotationMotionTimeout.Q THEN
        M_SetProcessError(uiAxisIndex := GVL_AxisIndex.DamperRotation, eErrorCode := E_DamperErrorCode.MotionTimeout);
    END_IF;

ELSE
    IF
        ioAxisRotation.State.bDone
        OR
        (
            ABS(ioAxisRotation.Data.fActPosition - fTargetAngle)
            <= GVL_MotionConfig.stDamper.stRotation.fPositionTolerance
        )
    THEN
        bRotationCommandIssued := FALSE;
        fbRotationMotionTimeout(IN := FALSE, PT := GVL_MotionConfig.stDamper.tMoveTimeout);
        M_MoveRotationAbsolute := TRUE;

    ELSIF ioAxisRotation.State.bCmdRejected THEN
        M_SetProcessError(uiAxisIndex := GVL_AxisIndex.DamperRotation, eErrorCode := E_DamperErrorCode.MotionCommandRejected);
    ELSIF ioAxisRotation.State.bCommandAborted THEN
        M_SetProcessError(uiAxisIndex := GVL_AxisIndex.DamperRotation, eErrorCode := E_DamperErrorCode.MotionCommandAborted);
    ELSIF fbRotationMotionTimeout.Q THEN
        M_SetProcessError(uiAxisIndex := GVL_AxisIndex.DamperRotation, eErrorCode := E_DamperErrorCode.MotionTimeout);
    END_IF;
END_IF;
END_METHOD

//==============================================================
// 两根独立轴在同一扫描周期启动绝对运动。
//
// 两根轴的bDone可能出现在不同扫描周期，因此分别锁存。
// 如果某根轴已经在目标位置，则不向该轴发送运动命令。
//==============================================================
METHOD PRIVATE M_MoveXYParallel : BOOL

VAR_INPUT
    fTargetX : LREAL;
    fTargetY : LREAL;
END_VAR

VAR_IN_OUT
    ioAxisX : ST_AxisInterface;
    ioAxisY : ST_AxisInterface;
END_VAR
M_MoveXYParallel := FALSE;
IF bError OR bAbort OR bReset THEN
    RETURN;
END_IF;


//==============================================================
// 1. 首次进入时判断每根轴是否需要运动
//==============================================================
IF NOT bXYCommandIssued THEN
    bXDoneLatched :=
        ABS(ioAxisX.Data.fActPosition - fTargetX)
        <= GVL_MotionConfig.stDamper.fPositionTolerance;

    bYDoneLatched :=
        ABS(ioAxisY.Data.fActPosition - fTargetY)
        <= GVL_MotionConfig.stDamper.fPositionTolerance;


    // X轴尚未到位时发送绝对运动脉冲。
    IF NOT bXDoneLatched THEN
        ioAxisX.AutoSet.Position.fAbsolutePosition := fTargetX;
        ioAxisX.AutoSet.Position.fVelocity :=
            GVL_MotionConfig.stDamper.stX.fVelocity;

        ioAxisX.AutoCmd.bMoveAbs := TRUE;
    END_IF;


    // Y轴尚未到位时发送绝对运动脉冲。
    IF NOT bYDoneLatched THEN
        ioAxisY.AutoSet.Position.fAbsolutePosition := fTargetY;
        ioAxisY.AutoSet.Position.fVelocity :=
            GVL_MotionConfig.stDamper.stY.fVelocity;

        ioAxisY.AutoCmd.bMoveAbs := TRUE;
    END_IF;

    bXYCommandIssued := TRUE;
END_IF;


//==============================================================
// 2. 分别锁存X、Y完成信号
//==============================================================
fbXYMotionTimeout(IN := bXYCommandIssued, PT := GVL_MotionConfig.stDamper.tMoveTimeout);
IF bXYCommandIssued THEN
    IF ioAxisX.State.bDone THEN
        bXDoneLatched := TRUE;
    END_IF;

    IF ioAxisY.State.bDone THEN
        bYDoneLatched := TRUE;
    END_IF;


    // 两根轴全部到位后，返回TRUE。
    IF bXDoneLatched AND bYDoneLatched THEN
        bXYCommandIssued := FALSE;
        bXDoneLatched := FALSE;
        bYDoneLatched := FALSE;

        fbXYMotionTimeout(IN := FALSE, PT := GVL_MotionConfig.stDamper.tMoveTimeout);
        M_MoveXYParallel := TRUE;
    ELSIF NOT ioAxisX.AutoCmd.bMoveAbs AND NOT ioAxisY.AutoCmd.bMoveAbs THEN
        // 双轴Done优先；否则任意轴Reject/Abort立即结束整个XY组。
        IF ioAxisX.State.bCmdRejected THEN
            M_SetProcessError(uiAxisIndex := GVL_AxisIndex.DamperX, eErrorCode := E_DamperErrorCode.MotionCommandRejected);
        ELSIF ioAxisY.State.bCmdRejected THEN
            M_SetProcessError(uiAxisIndex := GVL_AxisIndex.DamperY, eErrorCode := E_DamperErrorCode.MotionCommandRejected);
        ELSIF ioAxisX.State.bCommandAborted THEN
            M_SetProcessError(uiAxisIndex := GVL_AxisIndex.DamperX, eErrorCode := E_DamperErrorCode.MotionCommandAborted);
        ELSIF ioAxisY.State.bCommandAborted THEN
            M_SetProcessError(uiAxisIndex := GVL_AxisIndex.DamperY, eErrorCode := E_DamperErrorCode.MotionCommandAborted);
        ELSIF fbXYMotionTimeout.Q THEN
            IF NOT bXDoneLatched THEN
                M_SetProcessError(uiAxisIndex := GVL_AxisIndex.DamperX, eErrorCode := E_DamperErrorCode.MotionTimeout);
            ELSE
                M_SetProcessError(uiAxisIndex := GVL_AxisIndex.DamperY, eErrorCode := E_DamperErrorCode.MotionTimeout);
            END_IF;
        END_IF;
    END_IF;
END_IF;
END_METHOD

METHOD PRIVATE M_MoveZAbsolute : BOOL

VAR_INPUT
    fTargetZ : LREAL;
END_VAR

VAR_IN_OUT
    ioAxisZ : ST_AxisInterface;
END_VAR
M_MoveZAbsolute := FALSE;
IF bError OR bAbort OR bReset THEN
    RETURN;
END_IF;


//==============================================================
// 1. 发送一次Z轴绝对运动命令
//==============================================================
IF NOT bZCommandIssued THEN
    bZDoneLatched :=
        ABS(ioAxisZ.Data.fActPosition - fTargetZ)
        <= GVL_MotionConfig.stDamper.fPositionTolerance;

    IF NOT bZDoneLatched THEN
        ioAxisZ.AutoSet.Position.fAbsolutePosition := fTargetZ;
        ioAxisZ.AutoSet.Position.fVelocity :=
            GVL_MotionConfig.stDamper.stZ.fVelocity;

        ioAxisZ.AutoCmd.bMoveAbs := TRUE;
    END_IF;

    bZCommandIssued := TRUE;
END_IF;


//==============================================================
// 2. 等待运动完成
//==============================================================
fbZMotionTimeout(IN := bZCommandIssued, PT := GVL_MotionConfig.stDamper.tMoveTimeout);
IF bZCommandIssued THEN
    IF ioAxisZ.State.bDone THEN
        bZDoneLatched := TRUE;
    END_IF;

    IF bZDoneLatched THEN
        bZCommandIssued := FALSE;
        bZDoneLatched := FALSE;

        fbZMotionTimeout(IN := FALSE, PT := GVL_MotionConfig.stDamper.tMoveTimeout);
        M_MoveZAbsolute := TRUE;
    ELSIF NOT ioAxisZ.AutoCmd.bMoveAbs THEN
        IF ioAxisZ.State.bCmdRejected THEN
            M_SetProcessError(uiAxisIndex := GVL_AxisIndex.DamperZ, eErrorCode := E_DamperErrorCode.MotionCommandRejected);
        ELSIF ioAxisZ.State.bCommandAborted THEN
            M_SetProcessError(uiAxisIndex := GVL_AxisIndex.DamperZ, eErrorCode := E_DamperErrorCode.MotionCommandAborted);
        ELSIF fbZMotionTimeout.Q THEN
            M_SetProcessError(uiAxisIndex := GVL_AxisIndex.DamperZ, eErrorCode := E_DamperErrorCode.MotionTimeout);
        END_IF;
    END_IF;
END_IF;
END_METHOD

//==============================================================
// 从转台取回位取出已调整阻尼器，放到指定目标位置。
//
// 正常放回料盘时只需要改变fTargetX、fTargetY；
// fTargetZ固定传入fTrayPickZ。
//==============================================================
METHOD PRIVATE M_PlaceDamper : BOOL

VAR_INPUT
    fTargetX : LREAL;
    fTargetY : LREAL;
    fTargetZ : LREAL;
    fTargetSafeZ : LREAL;
END_VAR

VAR_IN_OUT
    ioAxisX : ST_AxisInterface;
    ioAxisY : ST_AxisInterface;
    ioAxisZ : ST_AxisInterface;
END_VAR
M_PlaceDamper := FALSE;

CASE ePlaceStep OF

    E_DamperPlaceStep.Idle:
        ePlaceStep :=
            E_DamperPlaceStep.EnsureTransferSafeZ;


    // 无论机械手当前在哪里，先确保Z轴到安全高度。
    E_DamperPlaceStep.EnsureTransferSafeZ:
        IF M_MoveZAbsolute(
            fTargetZ := fTransferSafeZ,
            ioAxisZ := ioAxisZ
        ) THEN
            ePlaceStep :=
                E_DamperPlaceStep.MoveXYToTransfer;
        END_IF;


    // 移动到转台取回位。
    E_DamperPlaceStep.MoveXYToTransfer:
        IF M_MoveXYParallel(
            fTargetX := fTransferX,
            fTargetY := fTransferY,
            ioAxisX := ioAxisX,
            ioAxisY := ioAxisY
        ) THEN
            ePlaceStep :=
                E_DamperPlaceStep.LowerZToTransfer;
        END_IF;


    // 下降到转台取回高度8mm。
    E_DamperPlaceStep.LowerZToTransfer:
        IF M_MoveZAbsolute(
            fTargetZ := fTransferPickZ,
            ioAxisZ := ioAxisZ
        ) THEN
            ePlaceStep :=
                E_DamperPlaceStep.ClampPlaceholder;
        END_IF;


    // 夹爪夹紧占位。
	// DamperZ已下降至转台取回高度。
	// 请求COM3夹爪夹紧；只有本次动作完成，才允许Z带料抬升。
	E_DamperPlaceStep.ClampPlaceholder:
		bGripperActionExecute := TRUE;
		eGripperActionCommand := E_GripperCommand.Close;
	
		// FB_GripperAction负责锁存本次请求编号，并验证有效反馈及bClosed。
		// Error由MAIN转入现有流程中止/全轴停止路径；本步骤不得继续。
		IF bGripperActionDone AND NOT bGripperActionError THEN
			ePlaceStep := E_DamperPlaceStep.LiftZFromTransfer;
		END_IF;

    // 从转台取回位升到15mm。
    E_DamperPlaceStep.LiftZFromTransfer:
        IF M_MoveZAbsolute(
            fTargetZ := fTransferSafeZ,
            ioAxisZ := ioAxisZ
        ) THEN
            ePlaceStep :=
                E_DamperPlaceStep.MoveXYToTarget;
        END_IF;


    // X、Y同时移动到调用方传入的目标坐标。
    E_DamperPlaceStep.MoveXYToTarget:
        IF M_MoveXYParallel(
            fTargetX := fTargetX,
            fTargetY := fTargetY,
            ioAxisX := ioAxisX,
            ioAxisY := ioAxisY
        ) THEN
            ePlaceStep :=
                E_DamperPlaceStep.LowerZToTarget;
        END_IF;


    // 下降到目标取放高度。
    E_DamperPlaceStep.LowerZToTarget:
        IF M_MoveZAbsolute(
            fTargetZ := fTargetZ,
            ioAxisZ := ioAxisZ
        ) THEN
            ePlaceStep :=
                E_DamperPlaceStep.ReleasePlaceholder;
        END_IF;


    // 夹爪松开占位。
	// DamperZ已下降至料盘目标位或最终缓冲位的放料高度。
	// 请求COM3夹爪张开；确认本次Open完成后才允许Z抬升。
	E_DamperPlaceStep.ReleasePlaceholder:
		bGripperActionExecute := TRUE;
		eGripperActionCommand := E_GripperCommand.Open;
	
		IF bGripperActionDone AND NOT bGripperActionError THEN
			ePlaceStep := E_DamperPlaceStep.LiftZFromTarget;
		END_IF;

    // 放料完成后回到目标安全高度。
    E_DamperPlaceStep.LiftZFromTarget:
        IF M_MoveZAbsolute(
            fTargetZ := fTargetSafeZ,
            ioAxisZ := ioAxisZ
        ) THEN
            ePlaceStep :=
                E_DamperPlaceStep.Completed;
        END_IF;


    E_DamperPlaceStep.Completed:
        M_PlaceDamper := TRUE;
        ePlaceStep := E_DamperPlaceStep.Idle;


ELSE
    ePlaceStep := E_DamperPlaceStep.Idle;

END_CASE;
END_METHOD

//==============================================================
// 初始化当前工作料盘的24个物理料位状态
//
// 新原材料料盘默认每个料位都放有未调整阻尼器。
//==============================================================
METHOD PRIVATE M_ResetDamperSlotStates

VAR
    nRow : DINT;
    nColumn : DINT;
END_VAR
//==============================================================
// 将4×6共24个料位全部设置为“未调整”。
// 本Method只修改状态，不修改料位坐标。
//==============================================================
FOR nRow := 1 TO UPPER_BOUND(aSlots, 1) DO
    FOR nColumn := 1 TO UPPER_BOUND(aSlots, 2) DO
        aSlots[nRow, nColumn].eState :=
            E_DamperSlotState.Unadjusted;
    END_FOR
END_FOR;
END_METHOD

METHOD PRIVATE M_ResetMotionHelpers

VAR_IN_OUT
    ioAxisX : ST_AxisInterface;
    ioAxisY : ST_AxisInterface;
    ioAxisZ : ST_AxisInterface;
	ioAxisRotation : ST_AxisInterface;
END_VAR
fbXYMotionTimeout(IN := FALSE, PT := GVL_MotionConfig.stDamper.tMoveTimeout);
fbZMotionTimeout(IN := FALSE, PT := GVL_MotionConfig.stDamper.tMoveTimeout);
fbRotationMotionTimeout(IN := FALSE, PT := GVL_MotionConfig.stDamper.tMoveTimeout);

// 复位XY并行运动内部状态
bXYCommandIssued := FALSE;
bXDoneLatched := FALSE;
bYDoneLatched := FALSE;

// 复位Z轴运动内部状态
bZCommandIssued := FALSE;
bZDoneLatched := FALSE;

// 清除可能残留的绝对运动命令
ioAxisX.AutoCmd.bMoveAbs := FALSE;
ioAxisY.AutoCmd.bMoveAbs := FALSE;
ioAxisZ.AutoCmd.bMoveAbs := FALSE;

// 复位单槽位Skip结果以及相机检测和旋转运行状态。
bTakeSkippedNoScrew := FALSE;
bTakeSkippedEmptySlot := FALSE;
fDetectedAngleLatched := 0.0;
fCorrectionAngleLatched := 0.0;
fRotationBaseAngle := GVL_PositionConfig.stDamper.fRotationZero;
fScanTargetAngle := GVL_PositionConfig.stDamper.fRotationZero;
bRotationCorrectionRequired := FALSE;
bRotationCommandIssued := FALSE;
// 复位夹紧后两个并行动作的完成锁存。
bCameraLiftZDoneLatched := FALSE;
bCameraRotationDoneLatched := FALSE;
// 复位放料后三个并行动作的完成锁存。
bResetLiftZDoneLatched := FALSE;
bResetTurntableDoneLatched := FALSE;
bResetRotationDoneLatched := FALSE;
// 清除可能残留的DamperRotation运动命令。
ioAxisRotation.AutoCmd.bMoveAbs := FALSE;
ioAxisRotation.AutoCmd.bMoveRel := FALSE;
END_METHOD

METHOD PRIVATE M_SetProcessError
VAR_INPUT
    uiAxisIndex : UINT;
    eErrorCode : E_DamperErrorCode;
END_VAR
// 仅锁存第一流程错误；Servo/NC/MC根因继续由Supervisor扫描轴报警。
IF NOT bError AND NOT bAbort AND NOT bReset THEN
    bError := TRUE;
    uiErrorAxis := uiAxisIndex;
    udiErrorCode := TO_UDINT(eErrorCode);
    eCurrentStep := E_DamperProcessStep.Error;
END_IF;
END_METHOD

//==============================================================
// 从指定料盘XY坐标取出未调整阻尼器，放入转台备料位。
//==============================================================
METHOD PRIVATE M_TakeDamper : BOOL

VAR_INPUT
    fSourceX : LREAL;
    fSourceY : LREAL;
END_VAR

VAR_IN_OUT
    ioAxisX : ST_AxisInterface;
    ioAxisY : ST_AxisInterface;
    ioAxisZ : ST_AxisInterface;
	// 阻尼器夹爪旋转轴。
    ioAxisRotation : ST_AxisInterface;
END_VAR
M_TakeDamper := FALSE;

CASE eTakeStep OF

    //==========================================================
    // 本次取料子流程开始
    //==========================================================
	E_DamperTakeStep.Idle:
		bTakeSkippedNoScrew := FALSE;
		bTakeSkippedEmptySlot := FALSE;
		// 清除上一件阻尼器锁存的视觉结果和机械角度基准。
		fDetectedAngleLatched := 0.0;
		fCorrectionAngleLatched := 0.0;
		fRotationBaseAngle := GVL_PositionConfig.stDamper.fRotationZero;
		fScanTargetAngle := GVL_PositionConfig.stDamper.fRotationZero;
		bRotationCorrectionRequired := FALSE;
		bVisionFault := FALSE;
		bVisionFallbackUsed := FALSE;
		eVisionError := E_VisionError.None;
	
		// 清除DamperRotation发令状态。
		bRotationCommandIssued := FALSE;
		// 清除两组并行动作完成锁存。
		bCameraLiftZDoneLatched := FALSE;
		bCameraRotationDoneLatched := FALSE;
		bResetLiftZDoneLatched := FALSE;
		bResetTurntableDoneLatched := FALSE;
		bResetRotationDoneLatched := FALSE;
	
		eTakeStep :=
			E_DamperTakeStep.EnsureSafeZ;

    //==========================================================
    // 1. 相机和XY移动前，先确保DamperZ位于110mm
    //==========================================================
    E_DamperTakeStep.EnsureSafeZ:
        IF M_MoveZAbsolute(
            fTargetZ := GVL_PositionConfig.stDamper.fSafeZ,
            ioAxisZ := ioAxisZ
        ) THEN
            eTakeStep :=
                E_DamperTakeStep.MoveXYToVisionPosition;
        END_IF;


    //==========================================================
    // 2. DamperXY移动，使相机中心对准当前阻尼器
    //
    // 相机位于夹爪Y正方向90mm：
    // 相机位置 = 夹爪位置 + 90mm
    //
    // 所以相机对准料位时：
    // 夹爪Y位置 = 料位Y位置 - 90mm
    //==========================================================
    E_DamperTakeStep.MoveXYToVisionPosition:
        fCurrentVisionX :=
            fSourceX - GVL_PositionConfig.stDamper.stCameraOffset.X;

        fCurrentVisionY :=
            fSourceY - GVL_PositionConfig.stDamper.stCameraOffset.Y;

        IF M_MoveXYParallel(
            fTargetX := fCurrentVisionX,
            fTargetY := fCurrentVisionY,
            ioAxisX := ioAxisX,
            ioAxisY := ioAxisY
        ) THEN
            eTakeStep :=
                E_DamperTakeStep.AcquireVisionResult;
        END_IF;


    //==========================================================
	// 3. 获取统一螺钉角度视觉结果
	//
	// Simulation与Camera均由FB_ScrewAngleVision返回相同强类型结果。
	// 视觉事务异常保持原锁存Error；正常有效但未检测到时只跳过当前槽位。
	//==========================================================
	E_DamperTakeStep.AcquireVisionResult:
		IF fbScrewAngleVision.bDone THEN
			// 两个角度语义保持独立；PLC不使用DetectedAngle计算机械修正量。
			fDetectedAngleLatched :=
				fbScrewAngleVision.stResult.fDetectedAngle;
			fCorrectionAngleLatched :=
				fbScrewAngleVision.stResult.fCorrectionAngle;
			fRotationBaseAngle := GVL_PositionConfig.stDamper.fRotationZero;
			bRotationCorrectionRequired := FALSE;

			bVisionFault := fbScrewAngleVision.bVisionFault;
			bVisionFallbackUsed := FALSE;
			eVisionError := fbScrewAngleVision.eVisionError;

			IF bVisionFault OR NOT fbScrewAngleVision.stResult.bValid THEN
				// 事务异常时绝不生成0度Fallback，也不进入后续取料、旋转和扫码流程。
				bVisionFault := TRUE;
				IF eVisionError = E_VisionError.None THEN
					eVisionError := E_VisionError.InvalidResult;
				END_IF;
				eTakeStep := E_DamperTakeStep.Idle;
				// Cancelled由整机主动终止产生，不新建Process Fault。
                CASE eVisionError OF
                    E_VisionError.Offline:
                        M_SetProcessError(uiAxisIndex := 0, eErrorCode := E_DamperErrorCode.ScrewVisionOffline);
                    E_VisionError.Timeout:
                        M_SetProcessError(uiAxisIndex := 0, eErrorCode := E_DamperErrorCode.ScrewVisionTimeout);
                    E_VisionError.ServiceFault:
                        M_SetProcessError(uiAxisIndex := 0, eErrorCode := E_DamperErrorCode.ScrewVisionServiceFault);
                    E_VisionError.TargetNotDetected:
                        M_SetProcessError(uiAxisIndex := 0, eErrorCode := E_DamperErrorCode.ScrewTargetNotDetected);
                    E_VisionError.Cancelled:
                        // Stop/Abort优先分支已撤销请求，不升级Cancelled。
                        bVisionFallbackUsed := FALSE;
                    ELSE
                        M_SetProcessError(uiAxisIndex := 0, eErrorCode := E_DamperErrorCode.ScrewVisionInvalidResult);
                END_CASE;
			ELSIF NOT fbScrewAngleVision.stResult.bDetected THEN
				// SkippedNoScrew：正常、有效、无故障结果；不等于物理空位。
				// 仅通知调用层推进搜索，绝不返回取料成功或建立回填目标。
				bTakeSkippedNoScrew := TRUE;
				eTakeStep := E_DamperTakeStep.Idle;
			ELSE
				// 仅CorrectionAngle参与机械控制；死区参数来自唯一ProcessConfig源。
				IF
					ABS(fCorrectionAngleLatched)
					> GVL_ProcessConfig.stVision.fAngleTolerance
				THEN
					fRotationBaseAngle :=
						GVL_PositionConfig.stDamper.fRotationZero
						+ fCorrectionAngleLatched;
					bRotationCorrectionRequired := TRUE;
				END_IF;

				// 旋转将在夹爪夹紧阻尼器后最多执行一次。
				bRotationCommandIssued := FALSE;
				bCameraRotationDoneLatched := FALSE;

				// 检测成功后，XY先回到理论料位。
				eTakeStep :=
					E_DamperTakeStep.MoveXYToSlot;
			END_IF;
		END_IF;


	//==========================================================
	// 4. 相机检测完成后，DamperXY回到阻尼器理论料位
	//
	// 此时只完成位置对准，DamperRotation暂不旋转。
	//==========================================================
    E_DamperTakeStep.MoveXYToSlot:
        IF M_MoveXYParallel(
            fTargetX := fSourceX,
            fTargetY := fSourceY,
            ioAxisX := ioAxisX,
            ioAxisY := ioAxisY
        ) THEN
            eTakeStep :=
                E_DamperTakeStep.LowerZToSlot;
        END_IF;


    // Z轴下降到当前设置的料盘取料绝对高度fTrayPickZ。
    E_DamperTakeStep.LowerZToSlot:
        IF M_MoveZAbsolute(
            fTargetZ := fTrayPickZ,
            ioAxisZ := ioAxisZ
        ) THEN
            eTakeStep :=
                E_DamperTakeStep.ClampPlaceholder;
        END_IF;


	//==========================================================
	// 6. 夹爪夹紧占位
	//
	// 当前没有接入阻尼器夹爪，直接认为夹紧完成。
	// 后续接入夹爪后，应在这里发送夹紧命令并等待夹紧反馈。
	//==========================================================
	E_DamperTakeStep.ClampPlaceholder:
		// DamperZ已到料盘取料高度。保持请求，动作FB仅在上升沿发一次Close。
		bGripperActionExecute := TRUE;
		eGripperActionCommand := E_GripperCommand.Close;
        bGripperAllowCloseTargetWithoutGrip := TRUE;
	
		// 本次Close被验证完成之前，禁止Z抬升和DamperRotation运动。
        IF bGripperActionDone AND NOT bGripperActionError THEN
            IF bGripperCloseTargetReachedWithoutGrip THEN
                // 唯一允许解释物理Empty的工艺位置；不建立虚拟工件。
                aSlots[nCurrentRow, nCurrentColumn].eState := E_DamperSlotState.Empty;
                bGripperActionExecute := FALSE;
                eGripperActionCommand := E_GripperCommand.None;
                bGripperAllowCloseTargetWithoutGrip := FALSE;
                eTakeStep := E_DamperTakeStep.EmptyReleaseClose;
            ELSE
                bCameraLiftZDoneLatched := FALSE;
                bCameraRotationDoneLatched := FALSE;
                bRotationCommandIssued := FALSE;
                eTakeStep := E_DamperTakeStep.RotationToCameraAngle;
            END_IF;
        END_IF;

    E_DamperTakeStep.EmptyReleaseClose:
        // Execute已释放；必须等Action Idle且旧Owner/Control Busy均已清除。
        // 本扫描仍不发Open，下一步才能形成独立Execute上升沿和RequestId。
        IF bGripperActionReady THEN
            eTakeStep := E_DamperTakeStep.EmptyOpen;
        END_IF;

    E_DamperTakeStep.EmptyOpen:
        bGripperActionExecute := TRUE;
        eGripperActionCommand := E_GripperCommand.Open;
        IF bGripperActionDone AND NOT bGripperActionError THEN
            bGripperActionExecute := FALSE;
            eGripperActionCommand := E_GripperCommand.None;
            eTakeStep := E_DamperTakeStep.EmptyLiftSafe;
        END_IF;

    E_DamperTakeStep.EmptyLiftSafe:
        // Open已完成；仅Z回现有安全高度，禁止XY/Rotation/扫码/交换。
        IF M_MoveZAbsolute(
            fTargetZ := GVL_PositionConfig.stDamper.fSafeZ,
            ioAxisZ := ioAxisZ
        ) THEN
            bTakeSkippedEmptySlot := TRUE;
            eTakeStep := E_DamperTakeStep.Idle;
        END_IF;
	//==========================================================
	// 7. Z轴抬升与DamperRotation绝对运动并行执行
	//
	// 同一个PLC扫描周期内：
	// 1. DamperZ开始向110mm安全位置运动；
	// 2. 仅当修正量超出死区时，DamperRotation绝对运动到修正后的机械基准角度。
	//
	// 两根轴分别锁存完成状态。
	// 只有两根轴全部完成后，XY才能移动到转台备料位。
	//==========================================================
	E_DamperTakeStep.RotationToCameraAngle:
	
		//======================================================
		// 7.1 启动并等待DamperZ抬升
		//======================================================
		IF NOT bCameraLiftZDoneLatched THEN
			IF M_MoveZAbsolute(
				fTargetZ := fTraySafeZ,
				ioAxisZ := ioAxisZ
			) THEN
				// Z轴完成信号可能只保持一个PLC周期，
				// 因此在这里锁存。
				bCameraLiftZDoneLatched := TRUE;
			END_IF;
		END_IF;
	
	
		//======================================================
		// 7.2 按需启动并等待DamperRotation单次角度修正
		//======================================================
		IF NOT bCameraRotationDoneLatched THEN
			IF NOT bRotationCorrectionRequired THEN
				// 修正量位于死区内，本件机械基准保持RotationZero，不发送旋转命令。
				bCameraRotationDoneLatched := TRUE;
			ELSIF M_MoveRotationAbsolute(
				fTargetAngle := fRotationBaseAngle,
				fVelocity := GVL_MotionConfig.stDamper.stRotation.fVelocity,
				fAcceleration := GVL_MotionConfig.stDamper.stRotation.fAcceleration,
				fDeceleration := GVL_MotionConfig.stDamper.stRotation.fDeceleration,
				ioAxisRotation := ioAxisRotation
			) THEN
				bCameraRotationDoneLatched := TRUE;
			END_IF;
		END_IF;
	
	
		//======================================================
		// 7.3 等待两个并行动作全部完成
		//======================================================
		IF
			bCameraLiftZDoneLatched
			AND bCameraRotationDoneLatched
		THEN
			// 清除本阶段并行运行状态。
			bCameraLiftZDoneLatched := FALSE;
			bCameraRotationDoneLatched := FALSE;
			bRotationCommandIssued := FALSE;
	
			// Z轴已经到达安全位置且本件角度修正已完成或无需修正，
			// 现在允许XY移动到转台备料位。
			eTakeStep :=
				E_DamperTakeStep.MoveXYToTransfer;
		END_IF;


	//==========================================================
	// 8. XY移动到转台备料位
	//
	// 此时DamperZ已经处于110mm安全高度。
	// XY到位后先执行二维码扫描，不立即下降Z轴。
	//==========================================================
	E_DamperTakeStep.MoveXYToTransfer:
		IF M_MoveXYParallel(
			fTargetX := fTransferX,
			fTargetY := fTransferY,
			ioAxisX := ioAxisX,
			ioAxisY := ioAxisY
		) THEN
			// 绝对扫码目标固定由本件实际机械基准角度与工艺偏移计算，
			// 不读取、不累加当前轴位置。
			fScanTargetAngle :=
				fRotationBaseAngle
				+ GVL_ProcessConfig.stQrScan.fOffsetAngle;
			bRotationCommandIssued := FALSE;
	
			eTakeStep :=
				E_DamperTakeStep.RotationToScanAngle;
		END_IF;
	//==========================================================
	// 9. DamperRotation绝对运动到扫码目标角度
	//
	// 当前机械状态：
	// 1. DamperX/Y已经到达转台备料位；
	// 2. DamperZ保持在110mm安全高度；
	// 3. 夹爪仍然夹持阻尼器。
	//
	// 当前二维码相机尚未接入，
	// DamperRotation到达“本件机械基准角度+扫码偏移角”即认为扫描成功。
	//==========================================================
	E_DamperTakeStep.RotationToScanAngle:
		IF M_MoveRotationAbsolute(
			fTargetAngle := fScanTargetAngle,
			fVelocity := GVL_MotionConfig.stDamperRotation.stQrScan.fVelocity,
			fAcceleration := GVL_MotionConfig.stDamperRotation.stQrScan.fAcceleration,
			fDeceleration := GVL_MotionConfig.stDamperRotation.stQrScan.fDeceleration,
			ioAxisRotation := ioAxisRotation
		) THEN
			// 扫码结束后允许DamperZ下降到备料取放高度。
			eTakeStep := E_DamperTakeStep.LowerZToTransfer;
		END_IF;
	// Z轴下降到实测备料位取放高度。
	// 当前fTransferPickZ为60mm。
    E_DamperTakeStep.LowerZToTransfer:
        IF M_MoveZAbsolute(
            fTargetZ := fTransferPickZ,
            ioAxisZ := ioAxisZ
        ) THEN
            eTakeStep :=
                E_DamperTakeStep.ReleasePlaceholder;
        END_IF;


    // 夹爪松开占位。
	E_DamperTakeStep.ReleasePlaceholder:
		// 已到备料位放料高度。确认本次Open完成后才允许Z抬升。
		bGripperActionExecute := TRUE;
		eGripperActionCommand := E_GripperCommand.Open;
	
		IF bGripperActionDone AND NOT bGripperActionError THEN
			// 工件已经实际放入备料位，先更新共享物料状态，
			// 但此时不启动转台；必须先确认DamperZ到达安全位置。
			eTransferPositionState := E_DamperSlotState.PendingAdjustment;
			stTurntableInput.bExchangeRequest := FALSE;
			stTurntableInput.bNoMorePartsToLoad := FALSE;

			bResetLiftZDoneLatched := FALSE;
			bResetTurntableDoneLatched := FALSE;
			bResetRotationDoneLatched := FALSE;
			bRotationCommandIssued := FALSE;

			eTakeStep := E_DamperTakeStep.RotationReturnHome;
		END_IF;

	//==========================================================
	// 10. 放料完成后的安全复位
	//
	// 第一阶段同时执行并分别锁存：
	// 1. DamperZ绝对运动到110mm安全高度；
	// 2. DamperRotation绝对运动到机械零点。
	//
	// 只有DamperZ确认到达安全高度后，才允许请求转台换位。
	//==========================================================
	E_DamperTakeStep.RotationReturnHome:
		IF NOT bResetLiftZDoneLatched THEN
			IF M_MoveZAbsolute(
				fTargetZ := fTransferSafeZ,
				ioAxisZ := ioAxisZ
			) THEN
				bResetLiftZDoneLatched := TRUE;
			END_IF;
		END_IF;

		IF NOT bResetRotationDoneLatched THEN
			IF M_MoveRotationAbsolute(
				fTargetAngle := GVL_PositionConfig.stDamper.fRotationZero,
				fVelocity := GVL_MotionConfig.stDamper.stRotation.fVelocity,
				fAcceleration := GVL_MotionConfig.stDamper.stRotation.fAcceleration,
				fDeceleration := GVL_MotionConfig.stDamper.stRotation.fDeceleration,
				ioAxisRotation := ioAxisRotation
			) THEN
				bResetRotationDoneLatched := TRUE;
			END_IF;
		END_IF;

		// Z轴安全到位是转台启动的唯一前置条件。
		// Rotation允许继续回零，不要求先于转台完成。
		IF bResetLiftZDoneLatched THEN
			stTurntableInput.bExchangeRequest := TRUE;
			stTurntableInput.bNoMorePartsToLoad := FALSE;

			eTakeStep := E_DamperTakeStep.WaitTurntableRotation;
		END_IF;

	//==========================================================
	// 11. Z轴已经安全到位，等待转台换位与Rotation回零
	//==========================================================
	E_DamperTakeStep.WaitTurntableRotation:
		// 如果Rotation回零尚未完成，继续执行并等待原绝对目标。
		IF NOT bResetRotationDoneLatched THEN
			IF M_MoveRotationAbsolute(
				fTargetAngle := GVL_PositionConfig.stDamper.fRotationZero,
				fVelocity := GVL_MotionConfig.stDamper.stRotation.fVelocity,
				fAcceleration := GVL_MotionConfig.stDamper.stRotation.fAcceleration,
				fDeceleration := GVL_MotionConfig.stDamper.stRotation.fDeceleration,
				ioAxisRotation := ioAxisRotation
			) THEN
				bResetRotationDoneLatched := TRUE;
			END_IF;
		END_IF;

		IF stTurntableStatus.bRotationDone THEN
			bResetTurntableDoneLatched := TRUE;
		END_IF;

		IF
			bResetLiftZDoneLatched
			AND bResetTurntableDoneLatched
			AND bResetRotationDoneLatched
		THEN
			bResetLiftZDoneLatched := FALSE;
			bResetTurntableDoneLatched := FALSE;
			bResetRotationDoneLatched := FALSE;
			bRotationCommandIssued := FALSE;

			eTakeStep := E_DamperTakeStep.Completed;
		END_IF;


    E_DamperTakeStep.Completed:
        M_TakeDamper := TRUE;
        eTakeStep := E_DamperTakeStep.Idle;


ELSE
    eTakeStep := E_DamperTakeStep.Idle;

END_CASE;
END_METHOD

END_FUNCTION_BLOCK

(* stored: Version 1.1.0.1, ProductVersion 3.1.4026.20
   POU FB_DamperProcess: Id {e2418071-795b-41d1-bc54-bf400327a8f1}, SpecialFunc None
   Method M_AbortProcess: Id {82b37050-c640-466e-b95e-c85810e5c597}
   Method M_InitializeDamperCoordinates: Id {cbc15f78-c68b-41b2-aed4-3f31228f7cac}
   Method M_MoveRotationAbsolute: Id {8b630280-4267-4fa1-8e7d-1778dc522e7e}
   Method M_MoveXYParallel: Id {76cd42f8-d1ed-4032-942b-c970dbafe1eb}
   Method M_MoveZAbsolute: Id {f9ca9d42-c75c-4515-95d3-d5d5d3ec6027}
   Method M_PlaceDamper: Id {0002ecd5-5e0f-4917-ab65-8cb804e7e274}
   Method M_ResetDamperSlotStates: Id {d593a935-7877-478b-9e7d-3d92c3c868b1}
   Method M_ResetMotionHelpers: Id {4692c3f6-cf16-4b48-9eab-0b11bbba2ad7}
   Method M_SetProcessError: Id {590f4f70-1358-4db5-b1f2-b05ddbdb0fec}
   Method M_TakeDamper: Id {d36fa61d-b49a-449e-ad76-302f3cdb0cc6} *)
